INTERFACE I_Cylinder

METHOD Extend
VAR_INPUT
END_VAR
END_METHOD

PROPERTY Extended : BOOL
GET
END_GET
END_PROPERTY

PROPERTY ExtendTime : LREAL
GET
END_GET
SET
END_SET
END_PROPERTY

METHOD Retract
VAR_INPUT
END_VAR
END_METHOD

PROPERTY Retracted : BOOL
GET
END_GET
END_PROPERTY

PROPERTY RetractTime : LREAL
GET
END_GET
SET
END_SET
END_PROPERTY

END_INTERFACE

(* stored: Version 1.1.0.1, ProductVersion 3.1.4024.15
   Itf I_Cylinder: Id {5eef6192-44e5-0f9f-3fe7-0d8e658e50b6}
   Method Extend: Id {6199c781-0269-09a7-1ca0-96654d2c0840}
   Property Extended: Id {9168958e-d017-0813-27ac-c9aa4feccc2e}
   Get Get: Id {02c5faf0-ce44-0130-0631-7cd44984288e}
   Property ExtendTime: Id {0500df96-c110-051e-1ea6-65dd24c85dea}
   Get Get: Id {a7fc8ac9-5ef2-03c5-075f-afa1154adfef}
   Set Set: Id {b68f8c8c-14dd-0bfe-0a28-814118c41844}
   Method Retract: Id {e7d61adf-37fc-023b-3604-04cdf6efdf9e}
   Property Retracted: Id {dde4e34a-b314-0277-079f-cf89835c0d08}
   Get Get: Id {4d086068-97be-0f17-0547-20f40cad0236}
   Property RetractTime: Id {37d15c05-fa62-0774-2651-73e0721efca8}
   Get Get: Id {add890c0-0961-0b40-1083-de218ca496fd}
   Set Set: Id {31e52a5b-921e-0a89-2d42-c41c36f5b9fd} *)
